(* PLC project Tc2_Utilities.UInt64Max Demo, tc3-libraries-kb TwinCAT 3.1 *)
(* stored: creationDateTime 2026-05-12T12:00:00, modificationDateTime 2026-05-12T12:00:00 *)

PROGRAM P_Demo_UInt64Max
  VAR
    uliA : T_ULARGE_INTEGER;;  (* 传感器 A 计数 *)
    uliB : T_ULARGE_INTEGER;;  (* 传感器 B 计数 *)
    uliMax : T_ULARGE_INTEGER;;  (* 较大者 *)
    bPick : BOOL;
  END_VAR

            // ============================================================
// Tc2_Utilities.UInt64Max 演示程序（FUNCTION，单周期触发）
// ============================================================
// 场景：多路温度传感器读回 64 位计数，取最大值做超温报警阈值比对。
// 价值：替代手写比较 + 选择；一次调用，可读性更高。
// 验证步骤：
//   1. 把本 PROGRAM 加到 PlcTask 调用列表
//   2. 编译 + 登录
//   3. 在线把 b... 触发位置 TRUE 一个周期
//   4. 观察输出变量是否符合期望
// ============================================================

IF bPick THEN
    uliMax := UInt64Max(uliA, uliB);
    bPick := FALSE;
END_IF;

          
END_PROGRAM
